PROGRAM MQTT_Subscriber
VAR
	
	received_msg_size : UDINT;
	sTopicSub : STRING;
	eQoSSub : TcIotMqttQos;
	bConnectSub : BOOL;
	MQTT_client : MQTTClient_Joints;	
	isConnected : BOOL;
	isSub : BOOL;
	
	joints_command AT %Q* : Joints;
	incoming_msg AT %I* : Joints;
END_VAR

sTopicSub := 'robot1/command'; 
eQoSSub := 1;
bConnectSub := TRUE;
isConnected := MQTT_client.bConnected;
MQTT_client.sHostName := '169.254.252.101';

//SUBSCRIBE
MQTT_client.Execute(bConnectSub);
isSub := MQTT_client.Subscribe(	sTopic := sTopicSub, 
								eQoS := eQoSSub);
incoming_msg := MQTT_client.sPayloadRcv;

joints_command := incoming_msg;

END_PROGRAM

(* stored: Version 1.1.0.1, ProductVersion 3.1.4024.10
   POU MQTT_Subscriber: Id {10df84a5-feb1-4676-a487-b177312612f8}, SpecialFunc None *)
